{attribute 'pack_mode' := '1'}
TYPE ST_EMAdsInput :
STRUCT
	sEMSensorPose				: ARRAY[1..4] OF S_EMSensorPose; // 下标=NDI通道号，未接入的通道为 0
    lError 						: LREAL;
    lDataScope 					: LREAL;
	bHeatBeat					: BOOL;// 心跳
END_STRUCT
END_TYPE

(* stored: Version 1.1.0.1, ProductVersion 3.1.4024.15
   DUT ST_EMAdsInput: Id {fd7acb80-875a-477a-b4db-9ab77ed07235} *)
